// TIA Portal V16 export
// export: Created 2022-11-17T11:55:26.5735308Z, ExportSetting WithDefaults, DisplayName Totally Integrated Automation Portal, DisplayVersion V16 Update 6, DisplayName TIA Portal Version Control Interface, DisplayVersion V16 Update 2, DisplayName TIA Portal Openness, DisplayVersion V16 Update 6, DisplayName SINAMICS Startdrive Advanced, DisplayVersion V16 Update 5, DisplayName SINAMICS Startdrive G130, G150, S120, S150, SINAMICS MV, S210, DisplayVersion V16 Update 5, DisplayName SINAMICS Startdrive G110M, G120, G120C, G120D, G120P, G115D, DisplayVersion V16 Update 5, DisplayName STEP 7 Professional, DisplayVersion V16 Update 6, DisplayName STEP 7 Safety, DisplayVersion V16, DisplayName WinCC Advanced, DisplayVersion V16 Update 6
DATA_BLOCK "DB09_TablePos"   // DB9
{ S7_Optimized_Access := 'FALSE' }
AUTHOR : Robopac
VERSION : 0.0
// stored: AutoNumber false, IsOnlyStoredInLoadMemory false, IsWriteProtectedInAS false
   VAR RETAIN
      dbx0_0 : Bool := FALSE;
      dbx0_1 : Bool := FALSE;
      dbx0_2 : Bool := TRUE;
      dbx0_3 : Bool := FALSE;
      dbx0_4 : Bool := FALSE;
      dbx0_5 : Bool := FALSE;
      dbx0_6 : Bool := FALSE;
      dbx0_7 : Bool := FALSE;
      dbx1_0 : Bool := FALSE;   // Table rotation axis movement forward
      dbx1_1 : Bool := FALSE;   // Table rotation axis movement backward
      dbx1_2 : Bool := FALSE;   // Table rotation axis movement inside low speed area
      dbx1_3 : Bool := FALSE;   // Table rotation axis movement low speed
      dbx1_4 : Bool := FALSE;   // Table rotation forward
      dbx1_5 : Bool := FALSE;   // Table rotation backward
      dbx1_6 : Bool := TRUE;
      dbx1_7 : Bool := FALSE;
      dbx2_0 : Bool := FALSE;
      dbx2_1 : Bool := FALSE;
      dbx2_2 : Bool := FALSE;
      dbx2_3 : Bool := FALSE;
      dbx2_4 : Bool := FALSE;
      dbx2_5 : Bool := FALSE;
      dbx2_6 : Bool := FALSE;
      dbx2_7 : Bool := FALSE;
      dbx3_0 : Bool := FALSE;   // Table rotation: Support for encoder running control
      dbx3_1 : Bool := FALSE;   // Table rotation: Support for encoder running control alarm
      dbx3_2 : Bool := FALSE;
      dbx3_3 : Bool := FALSE;
      dbx3_4 : Bool := FALSE;
      dbx3_5 : Bool := FALSE;
      dbx3_6 : Bool := FALSE;
      dbx3_7 : Bool := FALSE;
      dbx4_0 : Bool := FALSE;
      dbx4_1 : Bool := FALSE;
      dbx4_2 : Bool := FALSE;
      dbx4_3 : Bool := FALSE;
      dbx4_4 : Bool := FALSE;
      dbx4_5 : Bool := FALSE;
      dbx4_6 : Bool := FALSE;
      dbx4_7 : Bool := FALSE;
      dbx5_0 : Bool := FALSE;
      dbx5_1 : Bool := FALSE;
      dbx5_2 : Bool := FALSE;
      dbx5_3 : Bool := FALSE;
      dbw6 : Int := 5;   // Table rotation: Support for movement speed
      dbw8 : Int := 0;   // Table rotation: Support for movement deceleration
      dbw10 : Int := 5;   // Table rotation inverter: Support for speed selection
      dbw12 : Int := 10199;
      dbw14 : Int := 2340;
      dbw16 : Int := 0;
      dbw18 : Int := 0;
      dbw20 : Int := 0;
      dbw22 : Int := 0;
      dbw24 : Int := 0;
      dbw26 : Int := 0;
      dbw28 : Int := 0;
      dbd30 : DInt := -15;   // Table rotation position: Pulse
      dbw34 : Int := -8;   // Table position
      dbw36 : Int := 0;   // Table rotation position: Table maximum position
      dbw38 : Int := 0;   // Table rotation position: Deceleration position
      dbw40 : Int := 0;   // Table rotation position: Deceleration position
      dbd42 : DInt := -15;   // Support for encoder table rotation running control
      dbw46 : Int := 20;   // Support for encoder table rotation running control
      dbw48 : Int := -8;   // Table position according to offset
      dbw50 : Int := 0;
      dbw52 : Int := 0;
      dbw54 : Int := 0;
      dbw56 : Int := 0;
      dbw58 : Int := 0;
      dbw60 : Int := 0;
      dbw62 : Int := 0;
      dbw64 : Int := 0;
      dbw66 : Int := 0;
      dbw68 : Int := 0;
      dbw70 : Int := 0;
      Req1_Dest : Int := 0;   // Positioning request 1: Destination position
      Req2_Dest : Int := 0;   // Positioning request 2: Destination position
      Req3_Dest : Int := 0;   // Positioning request 3: Destination position
      Req4_Dest : Int := 0;   // Positioning request 4: Destination position
      Req1_Fwd : Bool := FALSE;   // Positioning request 1: Axis forward
      Req1_Bkw : Bool := FALSE;   // Positioning request 1: Axis backward
      Req1_Slow : Bool := FALSE;   // Positioning request 1: Axis slow speed
      Req1_Pos : Bool := FALSE;   // Positioning request 1: Axis in position
      Req2_Fwd : Bool := FALSE;   // Positioning request 2: Axis forward
      Req2_Bkw : Bool := FALSE;   // Positioning request 2: Axis backward
      Req2_Slow : Bool := FALSE;   // Positioning request 2: Axis slow speed
      Req2_Pos : Bool := FALSE;   // Positioning request 2: Axis in position
      Req3_Fwd : Bool := FALSE;   // Positioning request 3: Axis forward
      Req3_Bkw : Bool := FALSE;   // Positioning request 3: Axis backward
      Req3_Slow : Bool := FALSE;   // Positioning request 3: Axis slow speed
      Req3_Pos : Bool := FALSE;   // Positioning request 3: Axis in position
      Req4_Fwd : Bool := FALSE;   // Positioning request 4: Axis forward
      Req4_Bkw : Bool := FALSE;   // Positioning request 4: Axis backward
      Req4_Slow : Bool := FALSE;   // Positioning request 4: Axis slow speed
      Req4_Pos : Bool := FALSE;   // Positioning request 4: Axis in position
      Req5_Dest : Int := 0;   // Positioning request 4: Destination position
      Req6_Dest : Int := 0;   // Positioning request 4: Destination position
      Req7_Dest : Int := 0;   // Positioning request 4: Destination position
      Req8_Dest : Int := 0;   // Positioning request 4: Destination position
      Req5_Fwd : Bool := FALSE;   // Positioning request 5: Axis forward
      Req5_Bkw : Bool := FALSE;   // Positioning request 5: Axis backward
      Req5_Slow : Bool := FALSE;   // Positioning request 5: Axis slow speed
      Req5_Pos : Bool := FALSE;   // Positioning request 5: Axis in position
      Req6_Fwd : Bool := FALSE;   // Positioning request 6: Axis forward
      Req6_Bkw : Bool := FALSE;   // Positioning request 6: Axis backward
      Req6_Slow : Bool := FALSE;   // Positioning request 6: Axis slow speed
      Req6_Pos : Bool := FALSE;   // Positioning request 6: Axis in position
      Req7_Fwd : Bool := FALSE;   // Positioning request 7: Axis forward
      Req7_Bkw : Bool := FALSE;   // Positioning request 7: Axis backward
      Req7_Slow : Bool := FALSE;   // Positioning request 7: Axis slow speed
      Req7_Pos : Bool := FALSE;   // Positioning request 7: Axis in position
      Req8_Fwd : Bool := FALSE;   // Positioning request 8: Axis forward
      Req8_Bkw : Bool := FALSE;   // Positioning request 8: Axis backward
      Req8_Slow : Bool := FALSE;   // Positioning request 8: Axis slow speed
      Req8_Pos : Bool := FALSE;   // Positioning request 8: Axis in position
      dbw92 : Int := 0;
      dbw94 : Int := 0;
      dbw96 : Int := 0;
      dbw98 : Int := 0;
   END_VAR
BEGIN
END_DATA_BLOCK
